TYPE ST_ReceiveData :
STRUCT
	  Status      AT  %I*     : ST_ReceiveStatus;   
      Data        AT  %I*     : ARRAY[0..31]OF USINT;
END_STRUCT
END_TYPE

(* stored: Version 1.1.0.1, ProductVersion 3.1.4024.9
   DUT ST_ReceiveData: Id {3b3d10ea-a324-42a8-82a4-49619e46bbe3} *)
